(*********************************** G.D S.p.A. - Technical Department ***********************************
============= PROGRAM INFO ============
FOLDER:             TBD
MACHINES INVOLVED:  TBD 

============= DESCRIPTION =============
csp machine declaration

============= REVISIONS ===============
Date		Version	 	Author      	Description             
----------	-------		------------  	--------------------------------------------
2019/04/05 	0000.00	 	M.Grasso		Creation of the PRG

**********************************************************************************************************)
(*$R process_ref := prc; $*)
PROGRAM csp_case_feed_shuttle_accU
VAR
	
	prc:											process;
	prc_path:										STRING;
	
END_VAR

_read_var_input();

_object_manager();

IF NOT objects_running()
THEN
	RETURN;	
END_IF

_read_process_image();

_mode_manager();

_set_runtime_properties();

(********************************* BODY *********************************)
(************************************************************************)

_handle_messages();

_write_output();

ACTION _handle_messages:
;
END_ACTION

ACTION _handle_process_test:
;
END_ACTION

ACTION _mode_manager:
IF process_mode_req_is_pending(prc)
THEN
    process_apply_mode_req_first_step(prc);
    CASE process_get_mode(prc) OF
        MODE_TO_ABSENT:
			;
        MODE_TO_INACTIVE:
			;
        MODE_TO_TEST:
			;
        MODE_TO_OPERATIONAL:
			;
    END_CASE
    process_apply_mode_req_second_step(prc);
END_IF
END_ACTION

ACTION _object_manager:
IF objects_initialization()
THEN
	sub_process_init(
		object_name					:= 'csp_case_feed_shuttle_accU.prc', 
		process						:= csp_case_feed_shuttle.prc, 
		CONVERSION_this				:= prc);
		
	prc_path 						:= process_get_path(prc);
END_IF

IF objects_running()
THEN
	process_cycle(prc);
END_IF
END_ACTION

ACTION _read_process_image:
;
END_ACTION

ACTION _read_var_input:
;
END_ACTION

ACTION _set_runtime_properties:
;
END_ACTION

ACTION _write_output:
;
END_ACTION

END_PROGRAM

(* stored: Version 1.1.0.1, ProductVersion 3.1.4024.3
   POU csp_case_feed_shuttle_accU: Id {20285b63-6756-4d79-a1b6-7763c1f62766}, SpecialFunc None
   Action _handle_messages: Id {3f04f249-3fa5-4b87-b318-af1727aa4281}
   Action _handle_process_test: Id {27ac52fd-4dfa-4c8b-8d82-98095cbd0505}
   Action _mode_manager: Id {d01d51b9-e8dc-453b-8545-a30a723c4806}
   Action _object_manager: Id {a574a3f4-66f0-4f42-ae6b-a934504fa4fd}
   Action _read_process_image: Id {67dff22a-2f0d-43a0-b4ad-d64ba0308174}
   Action _read_var_input: Id {231e256a-e8b2-472a-8ec4-31fe38b27503}
   Action _set_runtime_properties: Id {85fbbbab-a22a-48e7-a055-0f76e656155d}
   Action _write_output: Id {a81bee43-df60-4636-a051-19118804d149} *)
